Omron CX-Programmer project NuevoProyecto (CX-Programmer 9.61)

# PLC P2E1V2: CJ2M CPU11

## Program NuevoPrograma1 (cyclic task 0)
Local symbols
Amarillo1 1.01 BOOL  ; 1.01
Amarillo2 1.09 BOOL  ; 1.09
Entrada1 0.00 BOOL  ; 0.00
Entrada2 0.01 BOOL  ; 0.01
Rojo1 1.00 BOOL  ; 1.00
Rojo2 1.08 BOOL  ; 1.08
Verde1 1.02 BOOL  ; 1.02
Verde2 1.10 BOOL  ; 1.10

### Section Sección1

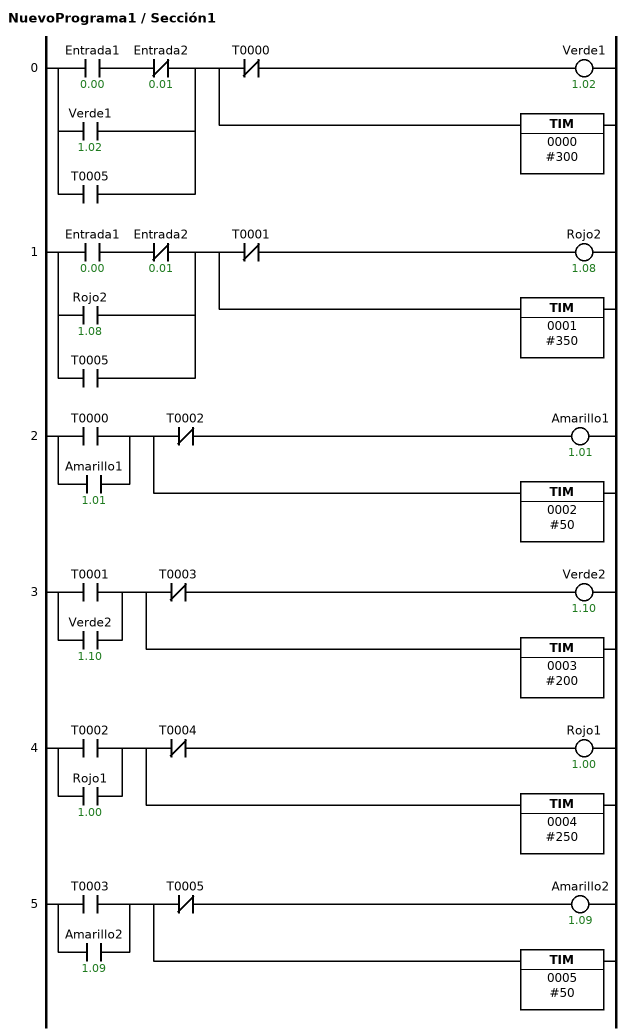
; rung 0
LD Entrada1  ; 0.00
ANDNOT Entrada2  ; 0.01
OR Verde1  ; 1.02
OR T0005
OUT TR0
ANDNOT T0000
OUT Verde1  ; 1.02
LD TR0
TIM 0000 #300
; rung 1
LD Entrada1  ; 0.00
ANDNOT Entrada2  ; 0.01
OR Rojo2  ; 1.08
OR T0005
OUT TR0
ANDNOT T0001
OUT Rojo2  ; 1.08
LD TR0
TIM 0001 #350
; rung 2
LD T0000
OR Amarillo1  ; 1.01
OUT TR0
ANDNOT T0002
OUT Amarillo1  ; 1.01
LD TR0
TIM 0002 #50
; rung 3
LD T0001
OR Verde2  ; 1.10
OUT TR0
ANDNOT T0003
OUT Verde2  ; 1.10
LD TR0
TIM 0003 #200
; rung 4
LD T0002
OR Rojo1  ; 1.00
OUT TR0
ANDNOT T0004
OUT Rojo1  ; 1.00
LD TR0
TIM 0004 #250
; rung 5
LD T0003
OR Amarillo2  ; 1.09
OUT TR0
ANDNOT T0005
OUT Amarillo2  ; 1.09
LD TR0
TIM 0005 #50

### Section END
; rung 0
END(001)